FUNCTION_BLOCK C_SERIALCOMM_PC EXTENDS C_SERIALCOMM_PORT
VAR_INPUT
END_VAR
VAR_OUTPUT
END_VAR
VAR
	_hwRxBuffer		AT %I* : PcComInData;
	_hwTxBuffer		AT %Q* : PcComOutData;
END_VAR

METHOD UPDATE_BUFFER : DINT
{message 'PC type Comm Port implemented'}
C_LINECONTROL(
	Mode:= SERIALLINEMODE_PC_COM_PORT, 
	pComIn:= ADR(_hwRxBuffer), 
	pComOut:= ADR(_hwTxBuffer), 
	SizeComIn:= SIZEOF(_hwRxBuffer), 
	TxBuffer:= _txbuffer, 
	RxBuffer:= _rxbuffer);
		
IF C_LINECONTROL.Error THEN
	UPDATE_BUFFER := 1;
	RETURN;
ELSE
	UPDATE_BUFFER := -1;
	RETURN;
END_IF
END_METHOD

END_FUNCTION_BLOCK

(* stored: Version 1.1.0.1, ProductVersion 3.1.4020.3
   POU C_SERIALCOMM_PC: Id {580a166b-08ad-475e-bc5e-6db98bee5c74}, SpecialFunc None
   Method UPDATE_BUFFER: Id {2b72e314-ba4c-4da8-8cfa-d4374b9c4505} *)
